Universal Robots PolyScope program: spiral.urp

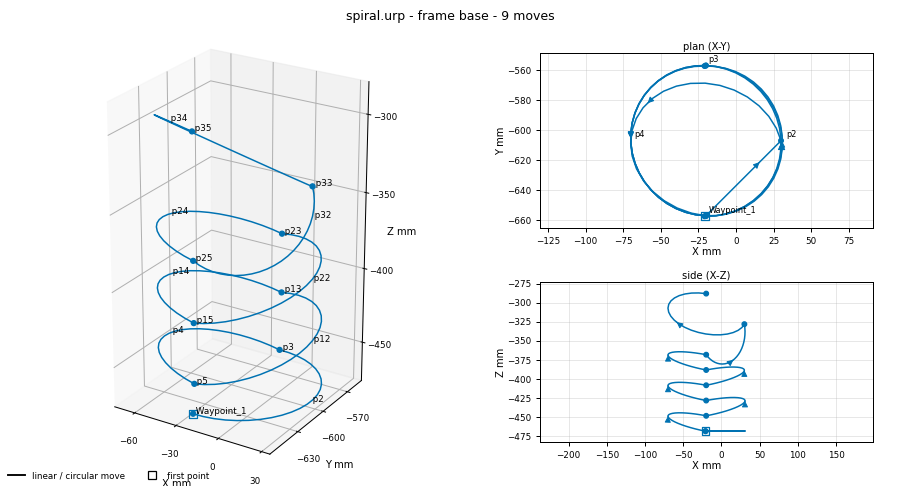
[picture p0: tool path of spiral.urp in frame base, 9 of 17 moves have a stored position in this frame; points joined in program order, loops and branches not executed]
Program spiral (installation=default directory=/home/ur/ursim-current/programs createdIn=5.12.6.1102099 lastSavedIn=5.12.6.1102099 robotSerialNumber=20195299999)
Calibrated DH parameters: a=[0, -0.6127, -0.57155, 0, 0, 0]; d=[0.1807, 0, 0, 0.17415, 0.11985, 0.11655]; alpha=[1.570796, 0, 0, 1.570796, -1.570796, 0]; deltaTheta=[0, 0, 0, 0, 0, 0]
Robot Program (runOnlyOnce=false)
  MoveP speed 250 mm/s, acceleration 1200 mm/s^2 (blendRadius=0.025 useActiveTCP=true) feature=Base
    Waypoint Waypoint_1: motionParameters(jointSpeed=1.047198 jointAcceleration=1.396263 cartesianSpeed=0.25 cartesianAcceleration=0.25); TCP in base x=-20.868 y=-657.352 z=-468.156 mm, rx=-0.0012 ry=3.1163 rz=0.0389 rad; joints [-76.78, -176.859, -102.636, 8.431, 91.725, 13.159] deg
    CircleMove (OrientationMode=UNCONSTRAINED)
      Waypoint p2: motionParameters(jointSpeed=1.047198 jointAcceleration=1.396263 cartesianSpeed=0.25 cartesianAcceleration=0.25); TCP in base x=30.87 y=-607.35 z=-468.156 mm, rx=-0.0012 ry=3.1163 rz=0.0389 rad; joints [-70.815, -177.952, -106.909, 13.982, 91.826, 19.126] deg
      Waypoint p3: motionParameters(jointSpeed=1.047198 jointAcceleration=1.396263 cartesianSpeed=0.25 cartesianAcceleration=0.25); TCP in base x=-20.87 y=-557.35 z=-468.156 mm, rx=-0.0012 ry=3.1163 rz=0.0389 rad; joints [-74.339, -179.504, -110.922, 19.436, 91.769, 15.601] deg
    CircleMove (OrientationMode=UNCONSTRAINED)
      Waypoint p4: TCP in base x=-70 y=-607.35 z=-448 mm, rx=-0.0012 ry=3.1163 rz=0.0389 rad; joints [-80.354, -175.884, -108.453, 13.167, 91.655, 9.585] deg
      Waypoint p5: TCP in base x=-20 y=-657 z=-448 mm, rx=-0.0012 ry=3.1163 rz=0.0389 rad; joints [-76.697, -174.954, -104.434, 8.325, 91.727, 13.242] deg
    CircleMove (OrientationMode=UNCONSTRAINED)
      Waypoint p12: TCP in base x=30.87 y=-607.35 z=-428 mm, rx=-0.0012 ry=3.1163 rz=0.0389 rad; joints [-70.815, -174.118, -110.45, 13.688, 91.826, 19.126] deg
      Waypoint p13: TCP in base x=-20 y=-557 z=-428 mm, rx=-0.0012 ry=3.1163 rz=0.0389 rad; joints [-74.238, -175.701, -114.587, 19.301, 91.771, 15.701] deg
    CircleMove (OrientationMode=UNCONSTRAINED)
      Waypoint p14: TCP in base x=-70 y=-607.35 z=-408 mm, rx=-0.0012 ry=3.1163 rz=0.0389 rad; joints [-80.354, -172.019, -111.868, 12.717, 91.655, 9.585] deg
      Waypoint p15: TCP in base x=-20 y=-657 z=-408 mm, rx=-0.0012 ry=3.1163 rz=0.0389 rad; joints [-76.697, -171.109, -107.772, 7.819, 91.727, 13.242] deg
    CircleMove (OrientationMode=UNCONSTRAINED)
      Waypoint p22: TCP in base x=30 y=-607 z=-388 mm, rx=-0.0012 ry=3.1163 rz=0.0389 rad; joints [-70.884, -170.214, -113.807, 13.139, 91.825, 19.057] deg
      Waypoint p23: TCP in base x=-20 y=-557 z=-388 mm, rx=-0.0012 ry=3.1163 rz=0.0389 rad; joints [-74.238, -171.78, -118.02, 18.813, 91.771, 15.701] deg
    CircleMove (OrientationMode=UNCONSTRAINED)
      Waypoint p24: TCP in base x=-70 y=-607 z=-368 mm, rx=-0.0012 ry=3.1163 rz=0.0389 rad; joints [-80.348, -168.062, -115.108, 12, 91.655, 9.59] deg
      Waypoint p25: TCP in base x=-20 y=-657 z=-368 mm, rx=-0.0012 ry=3.1163 rz=0.0389 rad; joints [-76.697, -167.188, -110.894, 7.019, 91.727, 13.242] deg
    CircleMove (OrientationMode=UNCONSTRAINED)
      Waypoint p32: TCP in base x=30 y=-607 z=-348 mm, rx=-0.0012 ry=3.1163 rz=0.0389 rad; joints [-70.884, -166.189, -116.925, 12.232, 91.825, 19.057] deg
      Waypoint p33: TCP in base x=30 y=-607 z=-328 mm, rx=-0.0012 ry=3.1163 rz=0.0389 rad; joints [-70.884, -164.13, -118.404, 11.652, 91.825, 19.057] deg
    CircleMove (OrientationMode=UNCONSTRAINED)
      Waypoint p34: TCP in base x=-70 y=-607 z=-308 mm, rx=-0.0012 ry=3.1163 rz=0.0389 rad; joints [-80.348, -161.889, -119.527, 10.245, 91.655, 9.59] deg
      Waypoint p35: TCP in base x=-20 y=-657 z=-288 mm, rx=-0.0012 ry=3.1163 rz=0.0389 rad; joints [-76.697, -159.069, -116.47, 4.477, 91.727, 13.242] deg
